// Mitsubishi GX Works2 project: PLC_Porject   PLC: FX3G

// global labels: Global1
VAR_GLOBAL CONSTANT
  counter_Time_2 : INT := K40;
END_VAR
VAR_GLOBAL
  init_reg AT M2 : BOOL;
END_VAR
VAR_GLOBAL CONSTANT
  choco_storage_input : REAL := 2000;
END_VAR
VAR_GLOBAL
  choco_stor_reg AT D1106 : REAL;
END_VAR
VAR_GLOBAL CONSTANT
  whip_storage_input : REAL := 2000;
END_VAR
VAR_GLOBAL
  whip_stor_reg AT D1108 : REAL;
END_VAR
VAR_GLOBAL CONSTANT
  biscu_storage_input : REAL := 300.0;
END_VAR
VAR_GLOBAL
  biscu_stor_reg AT D1110 : REAL;
  start_day AT X007 : BOOL;
  light_work_day AT Y007 : BOOL;
END_VAR
VAR_GLOBAL CONSTANT
  chco_for_trail : REAL := 240.0;
END_VAR
VAR_GLOBAL
  chco_have_min AT M4 : BOOL;
END_VAR
VAR_GLOBAL CONSTANT
  whip_for_trail : REAL := 300.0;
END_VAR
VAR_GLOBAL
  whip_have_min AT M6 : BOOL;
END_VAR
VAR_GLOBAL CONSTANT
  biscu_for_trail : REAL := 6.0;
END_VAR
VAR_GLOBAL
  biscu_have_min AT M5 : BOOL;
  all_condition_fill AT M7 : BOOL;
  emerg_switch AT X005 : BOOL;
  transport_end AT M8 : BOOL;
  storage_full AT M0 : BOOL;
END_VAR
VAR_GLOBAL CONSTANT
  counter_Time_1 : INT := K40;
END_VAR
VAR_GLOBAL
  tc_flash_timer AT TC1 : BOOL;
  ts_flash_timer AT TS1 : BOOL;
  tc_light_0_flash AT TC201 : BOOL;
  ts_light_0_flash AT TS201 : BOOL;
  light_0 AT Y000 : BOOL;
  tc_light_1_flash AT TC202 : BOOL;
  ts_light_1_flash AT TS202 : BOOL;
  light_1 AT Y001 : BOOL;
  biscu_start_reg AT D1104 : REAL;
  whip_start_reg AT D1102 : REAL;
  choco_start_reg AT D1100 : REAL;
  fill_whip_tank AT X011 : BOOL;
  init_whip_fill AT M1 : BOOL;
  whip_work_tank_reg AT D1112 : REAL;
  reset_flash AT M9 : BOOL;
  start_biscu_empty AT M3 : BOOL;
  start_whip_tank_empty AT M10 : BOOL;
  start_touch_sens AT X003 : BOOL;
  check_analog_input AT X006 : BOOL;
  analog_input_1 AT D8280 : INT;
END_VAR
VAR_GLOBAL CONSTANT
  LSL_regular_glaze : INT;
  LSL_double_glaze : INT := 2400;
END_VAR
VAR_GLOBAL
  regular_it_is AT Y005 : BOOL;
  double_it_is AT Y006 : BOOL;
END_VAR
VAR_GLOBAL CONSTANT
  choco_regular_for_trail : REAL := 120;
END_VAR
VAR_GLOBAL
  choco_work_tank_reg AT D1114 : REAL;
  tc_glazing_timer AT TC2 : BOOL;
  glazing_end AT M16 : BOOL;
  ts_glazing_timer AT TS2 : BOOL;
  ready_krembo AT D1210 : REAL;
  start_fill_tank_work_choco AT M18 : BOOL;
  machine_A_on AT Y004 : BOOL;
END_VAR
VAR_GLOBAL CONSTANT
  flash_time : INT := K40;
  USL_regular_glaze : INT := 2000;
END_VAR
VAR_GLOBAL
  regular_glaze AT M12 : BOOL;
END_VAR
VAR_GLOBAL CONSTANT
  USL_double_glaze : INT := 4000;
END_VAR
VAR_GLOBAL
  double_glaze AT M13 : BOOL;
END_VAR
VAR_GLOBAL CONSTANT
  glazing_time : INT := K50;
END_VAR
VAR_GLOBAL
  wrap_counter AT CC1 : BOOL;
  last_krembo_to_wrap AT Y002 : BOOL;
  wrap_one_krembo AT X000 : BOOL;
  five_krembo_wrapped AT CS1 : BOOL;
END_VAR
VAR_GLOBAL CONSTANT
  krembo_wrapped : INT := 5;
END_VAR
VAR_GLOBAL
  last_wrap_counter AT CC2 : BOOL;
  last_krembo_wrapped AT CS2 : BOOL;
  finished_wrapping AT M17 : BOOL;
  machine_B_on AT Y003 : BOOL;
  start_machine_A AT X010 : BOOL;
END_VAR
VAR_GLOBAL CONSTANT
  one_krembo_wrapped : INT := 2;
END_VAR
VAR_GLOBAL
  start_camera_sens AT X004 : BOOL;
  start_temp_sens_under_30 AT X002 : BOOL;
  start_temp_sens_under_15 AT X001 : BOOL;
END_VAR
VAR_GLOBAL CONSTANT
  empty_choco_work_tank : REAL;
END_VAR
VAR_GLOBAL
  check_tanks AT M19 : BOOL;
  help_check_tanks AT M20 : BOOL;
  end_day_reset_flash AT M21 : BOOL;
  flashed_three_time AT CS3 : BOOL;
  ts_end_flash_timer_on AT TS203 : BOOL;
  tc_end_flash_timer_on AT TC203 : BOOL;
END_VAR
VAR_GLOBAL CONSTANT
  ending_flash_time : INT := 80;
END_VAR
VAR_GLOBAL
  tc_end_flash_timer_off AT TC204 : BOOL;
  ts_end_flash_timer_off AT TS204 : BOOL;
  flash_counter AT CC3 : BOOL;
END_VAR
VAR_GLOBAL CONSTANT
  end_flashing_times : INT := 4;
END_VAR
VAR_GLOBAL
  first_itiration_ends AT M22 : BOOL;
  krembo_counter_2 AT CN2 : INT;
  krembo_counter_1 AT CN1 : INT;
END_VAR
VAR_GLOBAL CONSTANT
  empty_whip_work_tank : REAL;
END_VAR
VAR_GLOBAL
  analog_output AT D8282 : INT;
END_VAR
VAR_GLOBAL CONSTANT
  analog_output_cast : INT := 40;
  empty_ready_krembo_reg : REAL;
  empty_analog_output : INT;
END_VAR

// task Task_01 (event TRUE, interval 0, priority 31): POU_01

PROGRAM POU_01
(* structured ladder/FBD written out as ST: instructions are called as NAME(EN, inputs, outputs); _pN, _eN, _tN stand for wires *)
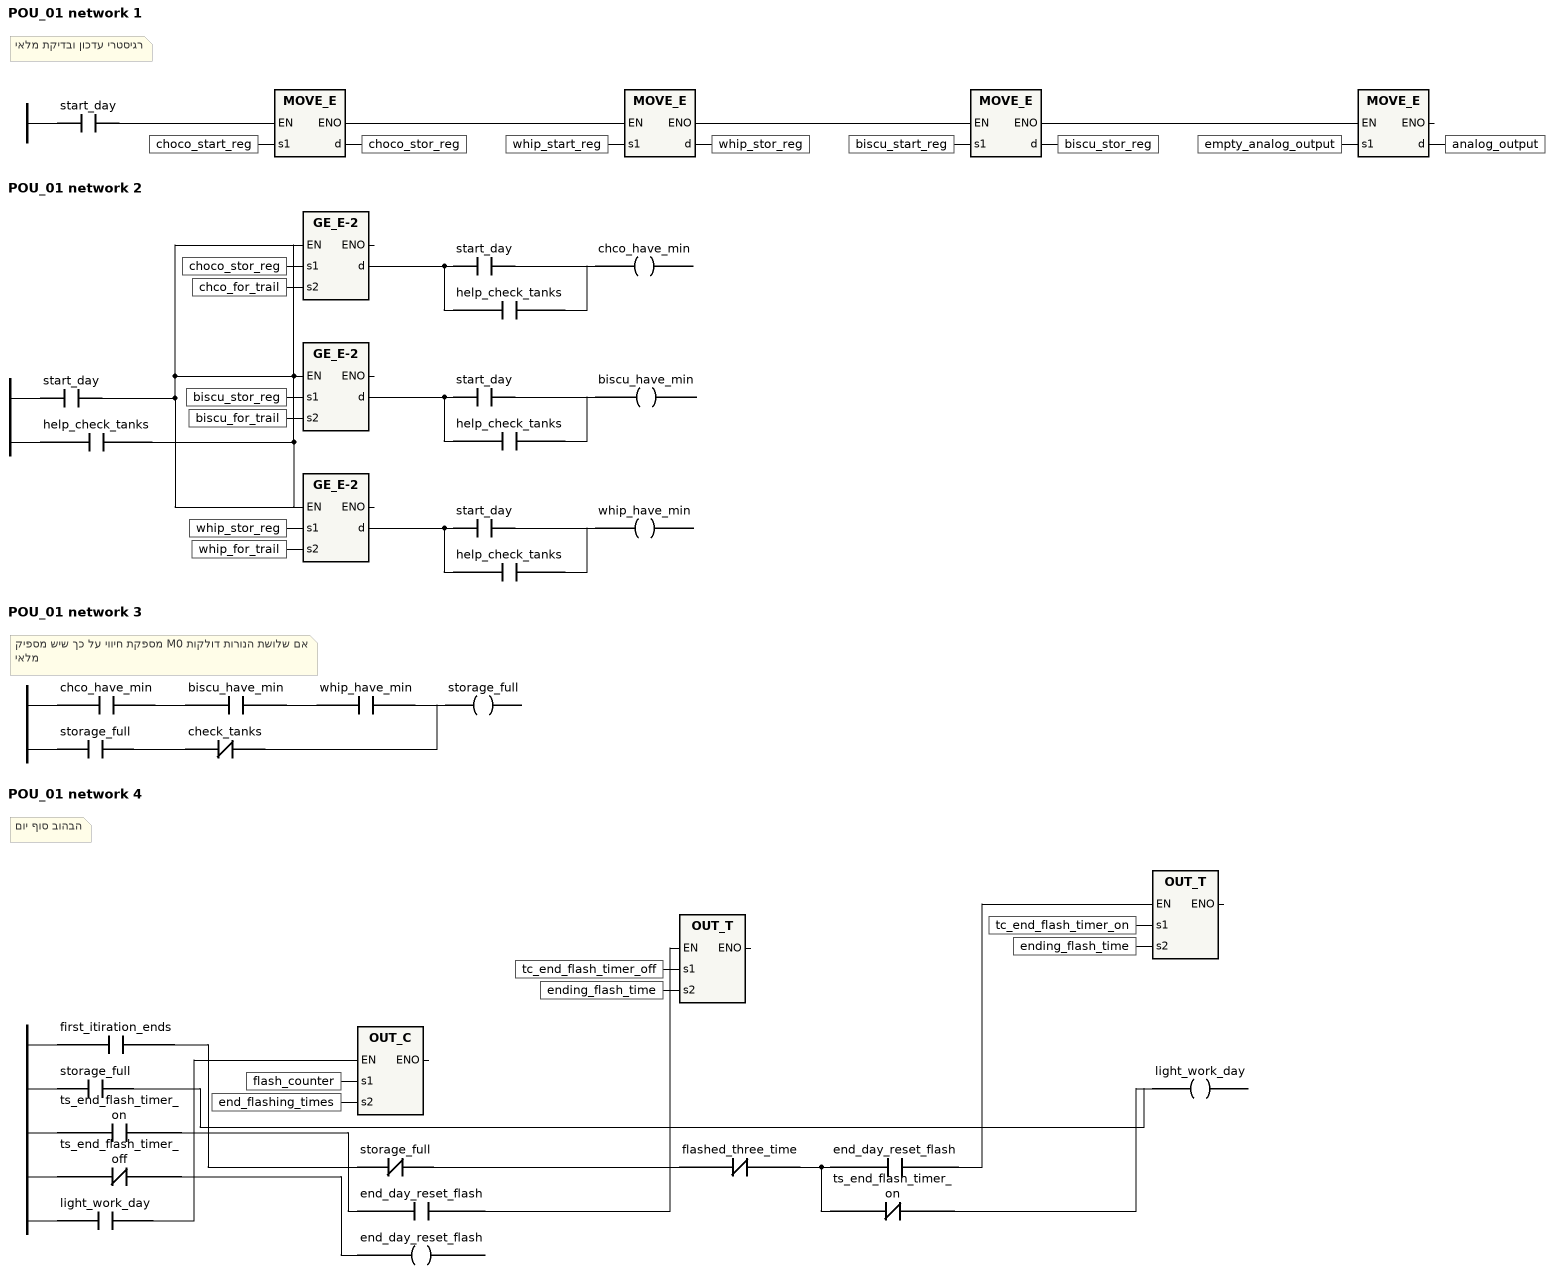
(* network 1 *)
(* רגיסטרי עדכון ובדיקת מלאי *)
_e1 := MOVE_E(start_day, choco_start_reg, choco_stor_reg);
_e2 := MOVE_E(_e1, whip_start_reg, whip_stor_reg);
_e3 := MOVE_E(_e2, biscu_start_reg, biscu_stor_reg);
MOVE_E(_e3, empty_analog_output, analog_output);
(* network 2 *)
_p1 := start_day OR help_check_tanks;
GE_E(_p1, choco_stor_reg, chco_for_trail, _t2);
chco_have_min := (_t2 AND start_day) OR (_t2 AND help_check_tanks);
GE_E(_p1, biscu_stor_reg, biscu_for_trail, _t3);
biscu_have_min := (_t3 AND start_day) OR (_t3 AND help_check_tanks);
GE_E(_p1, whip_stor_reg, whip_for_trail, _t4);
whip_have_min := (_t4 AND start_day) OR (_t4 AND help_check_tanks);
(* network 3 *)
(* אם שלושת הנורות דולקות M0 מספקת חיווי על כך שיש מספיק מלאי *)
storage_full := (chco_have_min AND biscu_have_min AND whip_have_min) OR (storage_full AND NOT check_tanks);
(* network 4 *)
(* הבהוב סוף יום *)
_p1 := first_itiration_ends AND NOT storage_full AND NOT flashed_three_time;
OUT_T(_p1 AND end_day_reset_flash, tc_end_flash_timer_on, ending_flash_time);
light_work_day := (_p1 AND NOT ts_end_flash_timer_on) OR storage_full;
OUT_T(ts_end_flash_timer_on AND end_day_reset_flash, tc_end_flash_timer_off, ending_flash_time);
end_day_reset_flash := NOT ts_end_flash_timer_off;
OUT_C(light_work_day, flash_counter, end_flashing_times);
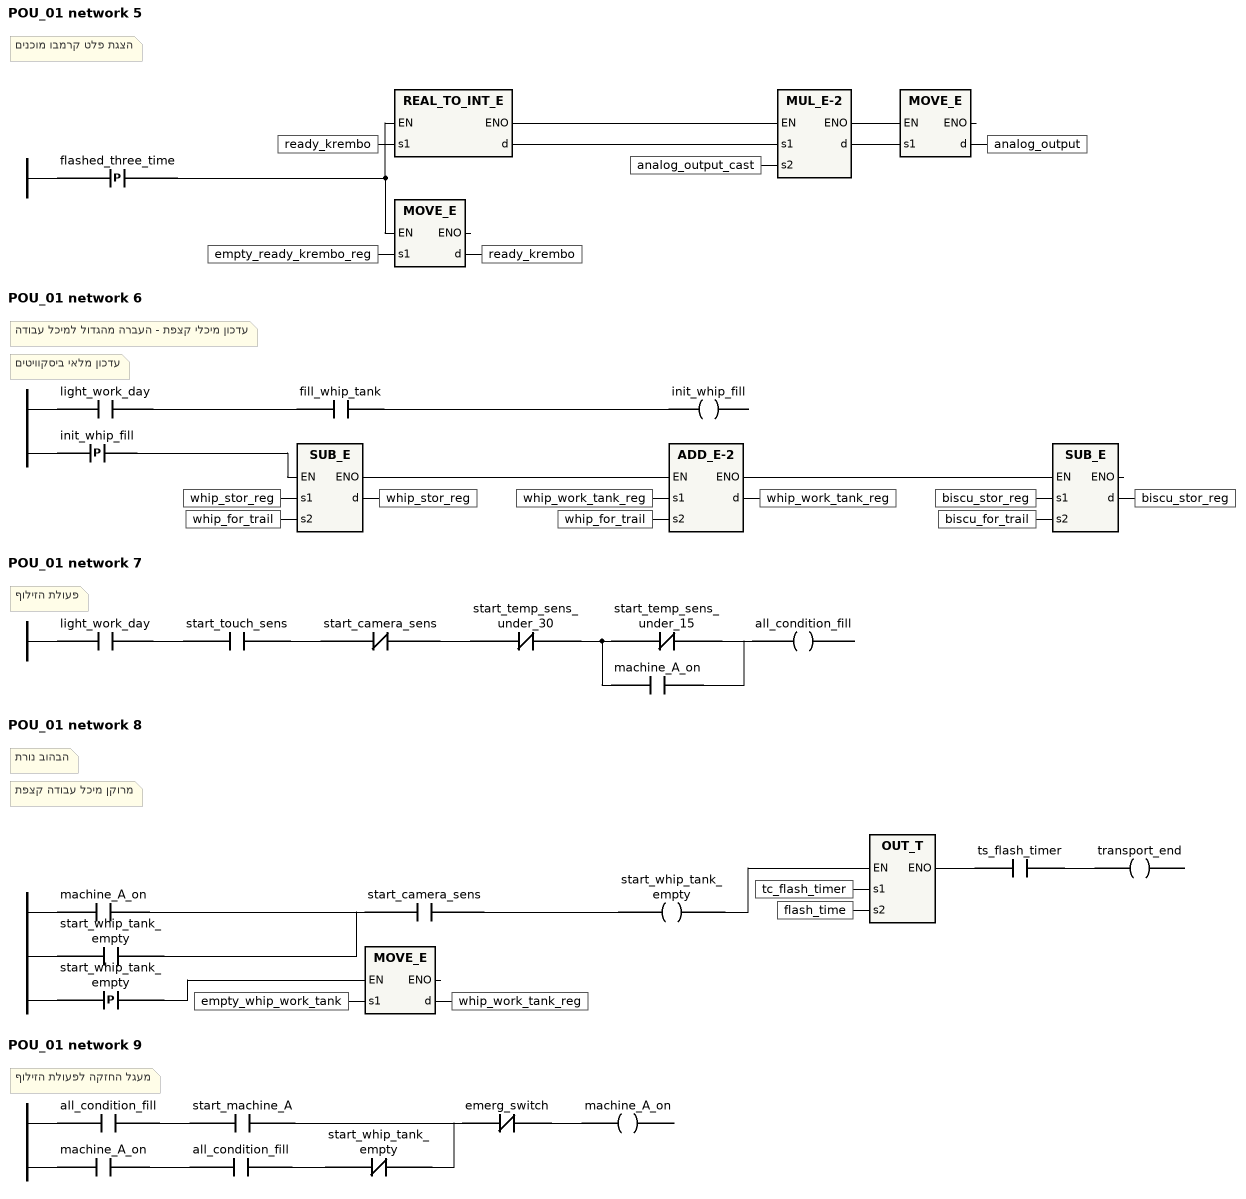
(* network 5 *)
(* הצגת פלט קרמבו מוכנים *)
_p1 := LDP(TRUE, flashed_three_time);
_e3 := REAL_TO_INT_E(_p1, ready_krembo, _t2);
_e5 := MUL_E(_e3, _t2, analog_output_cast, _t4);
MOVE_E(_e5, _t4, analog_output);
MOVE_E(_p1, empty_ready_krembo_reg, ready_krembo);
(* network 6 *)
(* עדכון מיכלי קצפת - העברה מהגדול למיכל עבודה *)
(* עדכון מלאי ביסקוויטים *)
init_whip_fill := light_work_day AND fill_whip_tank;
_e1 := SUB_E(LDP(TRUE, init_whip_fill), whip_stor_reg, whip_for_trail, whip_stor_reg);
_e2 := ADD_E(_e1, whip_work_tank_reg, whip_for_trail, whip_work_tank_reg);
SUB_E(_e2, biscu_stor_reg, biscu_for_trail, biscu_stor_reg);
(* network 7 *)
(* פעולת הזילוף *)
_p1 := light_work_day AND start_touch_sens AND NOT start_camera_sens AND NOT start_temp_sens_under_30;
all_condition_fill := (_p1 AND NOT start_temp_sens_under_15) OR (_p1 AND machine_A_on);
(* network 8 *)
(* הבהוב נורת *)
(* מרוקן מיכל עבודה קצפת *)
_p1 := (machine_A_on OR start_whip_tank_empty) AND start_camera_sens;
start_whip_tank_empty := _p1;
_e2 := OUT_T(_p1, tc_flash_timer, flash_time);
transport_end := _e2 AND ts_flash_timer;
MOVE_E(LDP(TRUE, start_whip_tank_empty), empty_whip_work_tank, whip_work_tank_reg);
(* network 9 *)
(* מעגל החזקה לפעולת הזילוף *)
machine_A_on := ((all_condition_fill AND start_machine_A) OR (machine_A_on AND all_condition_fill AND NOT start_whip_tank_empty)) AND NOT emerg_switch;
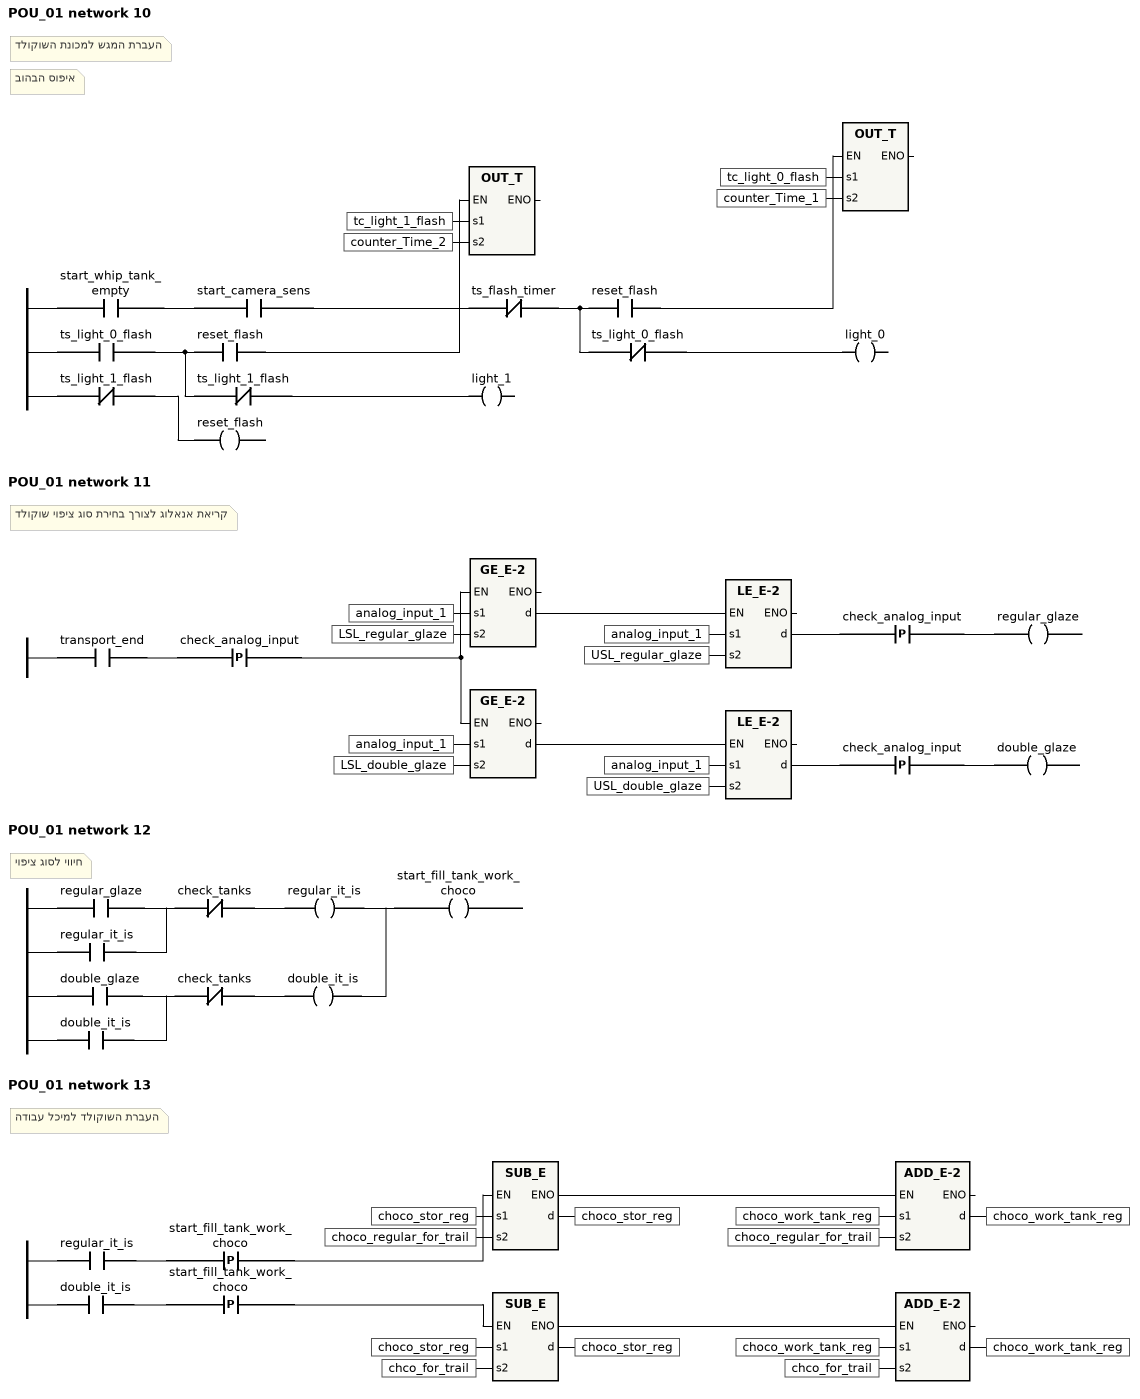
(* network 10 *)
(* העברת המגש למכונת השוקולד *)
(* איפוס הבהוב *)
_p1 := start_whip_tank_empty AND start_camera_sens AND NOT ts_flash_timer;
OUT_T(_p1 AND reset_flash, tc_light_0_flash, counter_Time_1);
light_0 := _p1 AND NOT ts_light_0_flash;
OUT_T(ts_light_0_flash AND reset_flash, tc_light_1_flash, counter_Time_2);
light_1 := ts_light_0_flash AND NOT ts_light_1_flash;
reset_flash := NOT ts_light_1_flash;
(* network 11 *)
(* קריאת אנאלוג לצורך בחירת סוג ציפוי שוקולד *)
_p1 := transport_end AND LDP(TRUE, check_analog_input);
GE_E(_p1, analog_input_1, LSL_regular_glaze, _t2);
LE_E(_t2, analog_input_1, USL_regular_glaze, _t3);
regular_glaze := _t3 AND LDP(TRUE, check_analog_input);
GE_E(_p1, analog_input_1, LSL_double_glaze, _t4);
LE_E(_t4, analog_input_1, USL_double_glaze, _t5);
double_glaze := _t5 AND LDP(TRUE, check_analog_input);
(* network 12 *)
(* חיווי לסוג ציפוי *)
_p1 := (regular_glaze OR regular_it_is) AND NOT check_tanks;
regular_it_is := _p1;
_p2 := (double_glaze OR double_it_is) AND NOT check_tanks;
double_it_is := _p2;
start_fill_tank_work_choco := _p1 OR _p2;
(* network 13 *)
(* העברת השוקולד למיכל עבודה *)
_e1 := SUB_E(regular_it_is AND LDP(TRUE, start_fill_tank_work_choco), choco_stor_reg, choco_regular_for_trail, choco_stor_reg);
ADD_E(_e1, choco_work_tank_reg, choco_regular_for_trail, choco_work_tank_reg);
_e2 := SUB_E(double_it_is AND LDP(TRUE, start_fill_tank_work_choco), choco_stor_reg, chco_for_trail, choco_stor_reg);
ADD_E(_e2, choco_work_tank_reg, chco_for_trail, choco_work_tank_reg);
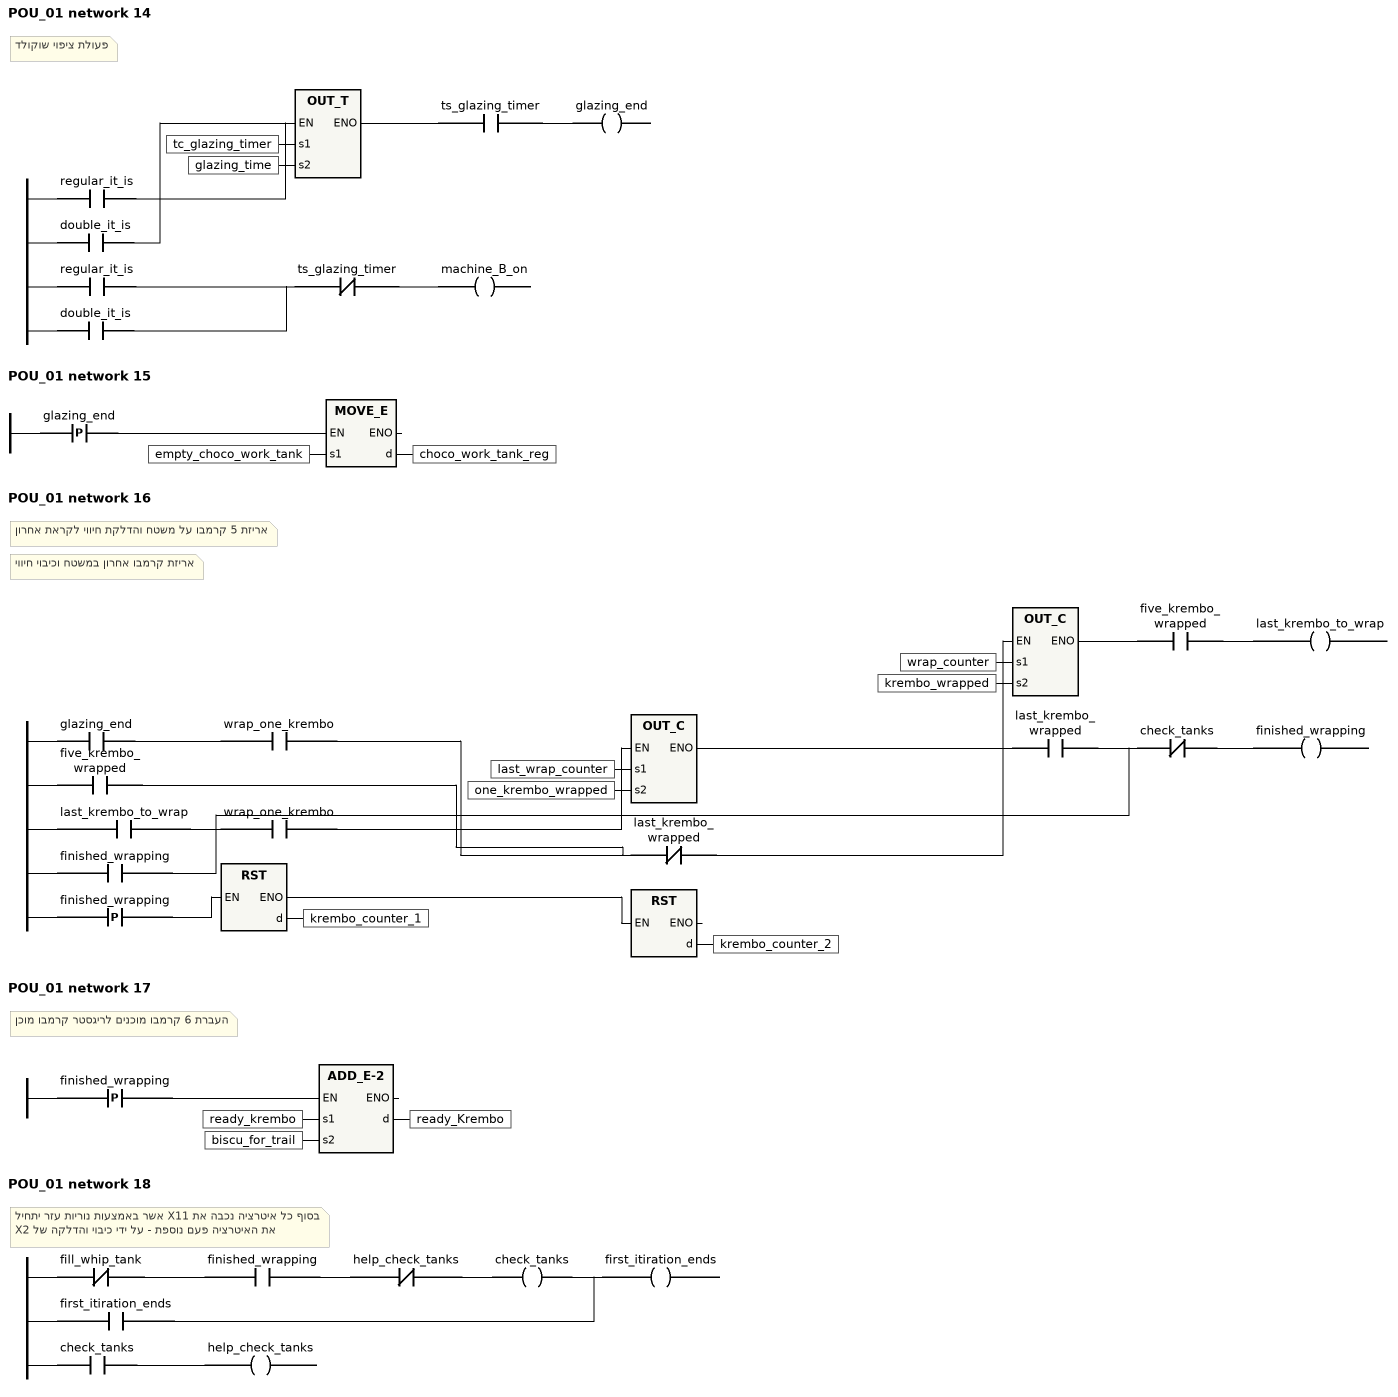
(* network 14 *)
(* פעולת ציפוי שוקולד *)
_e1 := OUT_T(regular_it_is OR double_it_is, tc_glazing_timer, glazing_time);
glazing_end := _e1 AND ts_glazing_timer;
machine_B_on := (regular_it_is OR double_it_is) AND NOT ts_glazing_timer;
(* network 15 *)
MOVE_E(LDP(TRUE, glazing_end), empty_choco_work_tank, choco_work_tank_reg);
(* network 16 *)
(* אריזת 5 קרמבו על משטח והדלקת חיווי לקראת אחרון *)
(* אריזת קרמבו אחרון במשטח וכיבוי חיווי *)
_e1 := OUT_C(((glazing_end AND wrap_one_krembo) OR five_krembo_wrapped) AND NOT last_krembo_wrapped, wrap_counter, krembo_wrapped);
last_krembo_to_wrap := _e1 AND five_krembo_wrapped;
_e2 := OUT_C(last_krembo_to_wrap AND wrap_one_krembo, last_wrap_counter, one_krembo_wrapped);
finished_wrapping := ((_e2 AND last_krembo_wrapped) OR finished_wrapping) AND NOT check_tanks;
_e3 := RST(LDP(TRUE, finished_wrapping), krembo_counter_1);
RST(_e3, krembo_counter_2);
(* network 17 *)
(* העברת 6 קרמבו מוכנים לריגסטר קרמבו מוכן *)
ADD_E(LDP(TRUE, finished_wrapping), ready_krembo, biscu_for_trail, ready_Krembo);
(* network 18 *)
(* בסוף כל איטרציה נכבה את X11 אשר באמצעות נוריות עזר יתחיל את האיטרציה פעם נוספת - על ידי כיבוי והדלקה של X2 *)
_p1 := NOT fill_whip_tank AND finished_wrapping AND NOT help_check_tanks;
check_tanks := _p1;
first_itiration_ends := _p1 OR first_itiration_ends;
help_check_tanks := check_tanks;
END_PROGRAM
